PROGRAM stopping_mode
VAR
	ed_routine_stopping_idle: BOOL;
	stack_power_enabled: BOOL;
	RECTIFIER_OUTPUT_OFF: BOOL;// ADD LOGIC FOR MONITORING RECTIFIER OUTPUT - USE CT? VERIFY PS DOES NOT MOVE CURRENT WHEN POWERED OFF
	u_3112_b_stop_request: BOOL;
	u_3212_b_stop_request: BOOL;
	u_3312_b_stop_request: BOOL;
	u_3405_b_stop_request: BOOL;
	u_3160_b_stop_request: BOOL
;
	u_3260_b_stop_request: BOOL;
	u_3360_b_stop_request: BOOL;
	u_3370_b_stop_request: BOOL;
	u_3112_b_run_feedback: BOOL;
	u_3212_b_run_feedback: BOOL;
	u_3312_b_run_feedback: BOOL;
	u_3405_b_run_feedback: BOOL;
	u_3160_b_run_feedback: BOOL;
	u_3260_b_run_feedback: BOOL;
	u_3360_b_run_feedback: BOOL;
	u_3370_b_run_feedback: BOOL;
	
	nv_3110_b_stop_request:BOOL;
	av_3248_b_stop_request: BOOL;
	av_3148_b_stop_request: BOOL;
	nv_3335_b_stop_request: BOOL;
	nv_3235_b_stop_request: BOOL;
	nv_3135_b_stop_request: BOOL;
	nv_3310_b_stop_request: BOOL;
	nv_3210_b_stop_request: BOOL;
	ed_routine_stop_mode: BOOL;
	redox_doser_stop_request: BOOL;
	nv_3335_b_position_request: INT;
	av_3148_b_position_request: INT;
	av_3248_b_position_request: INT;
	ed_pumps_stopped: BOOL;

	nv_3335_b_position_feedback: INT;
	nv_3335_b_recycle_position: BOOL;
	av_3148_b_position_feedback: INT;
	av_3148_b_recycle_position: BOOL;
	av_3248_b_recycle_position: BOOL;
	ed_valves_stopped: BOOL;
	ed_stopped: BOOL;
	av_3348_b_position_request: INT;
	nv_3372_b_stop_request: BOOL;
	av_3348_b_position_feedback: INT;
	av_3348_b_recycle_position: BOOL;
	nv_3335_b_closed_feedback: BOOL;
	nv_3372_b_closed_feedback: BOOL;
	nv_3162_b_stop_request: BOOL;
	ed_critical_stop: BOOL;
	tmr_stop_pump_delay: TON;
	tmr_stop_pump_delay_pt: TIME := T#10S;
	tmr_stop_pump_delay_et: TIME;
	test_ramp: ramp;
	eng_test: BOOL;
	test_ramp_start_val: REAL;
	test_ramp_end_val: REAL;
	test_ramp_duration: INT;
END_VAR
VAR // added by the converter: edge detectors and wires of the graphical bodies
    _w1, _w2, _w3 : BOOL;
END_VAR

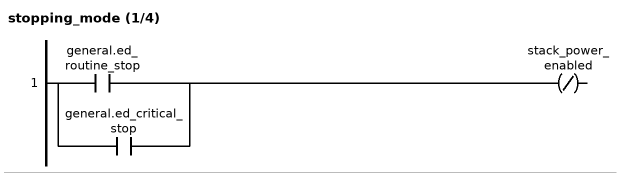
// NETWORK 1
stack_power_enabled := NOT (general.ed_routine_stop OR general.ed_critical_stop);

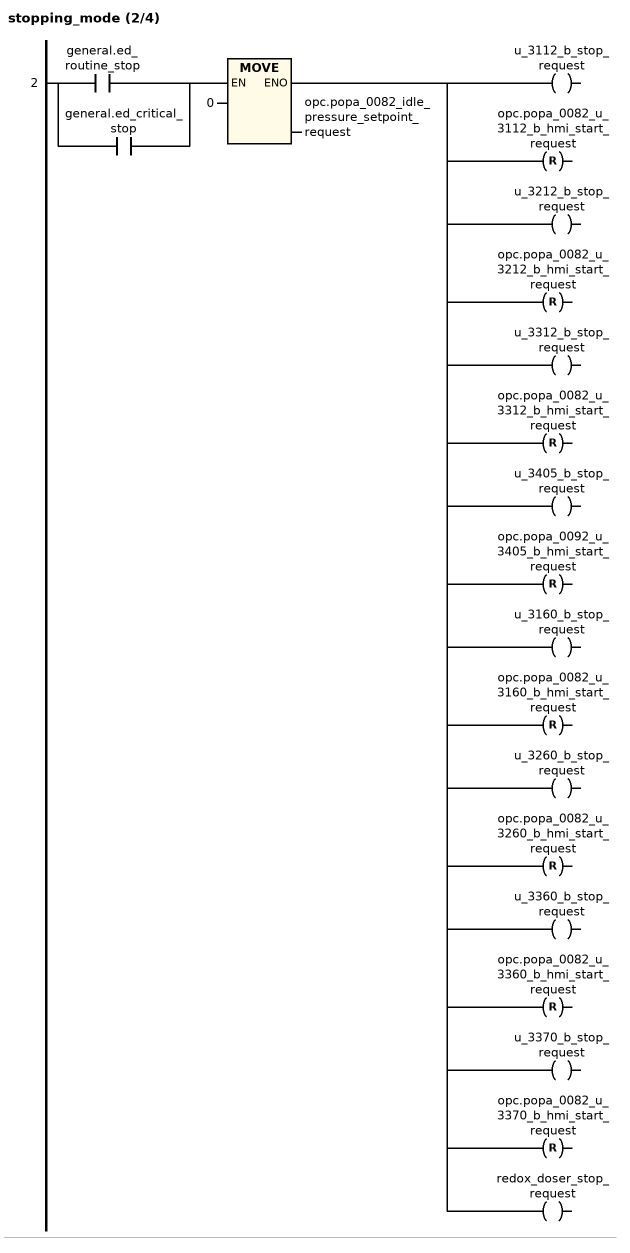
// NETWORK 2
_w1 := general.ed_routine_stop OR general.ed_critical_stop;
IF _w1 THEN opc.popa_0082_idle_pressure_setpoint_request := 0; END_IF
u_3112_b_stop_request := _w1;
opc.popa_0082_u_3112_b_hmi_start_request R= _w1;
u_3212_b_stop_request := _w1;
opc.popa_0082_u_3212_b_hmi_start_request R= _w1;
u_3312_b_stop_request := _w1;
opc.popa_0082_u_3312_b_hmi_start_request R= _w1;
u_3405_b_stop_request := _w1;
opc.popa_0092_u_3405_b_hmi_start_request R= _w1;
u_3160_b_stop_request := _w1;
opc.popa_0082_u_3160_b_hmi_start_request R= _w1;
u_3260_b_stop_request := _w1;
opc.popa_0082_u_3260_b_hmi_start_request R= _w1;
u_3360_b_stop_request := _w1;
opc.popa_0082_u_3360_b_hmi_start_request R= _w1;
u_3370_b_stop_request := _w1;
opc.popa_0082_u_3370_b_hmi_start_request R= _w1;
redox_doser_stop_request := _w1;

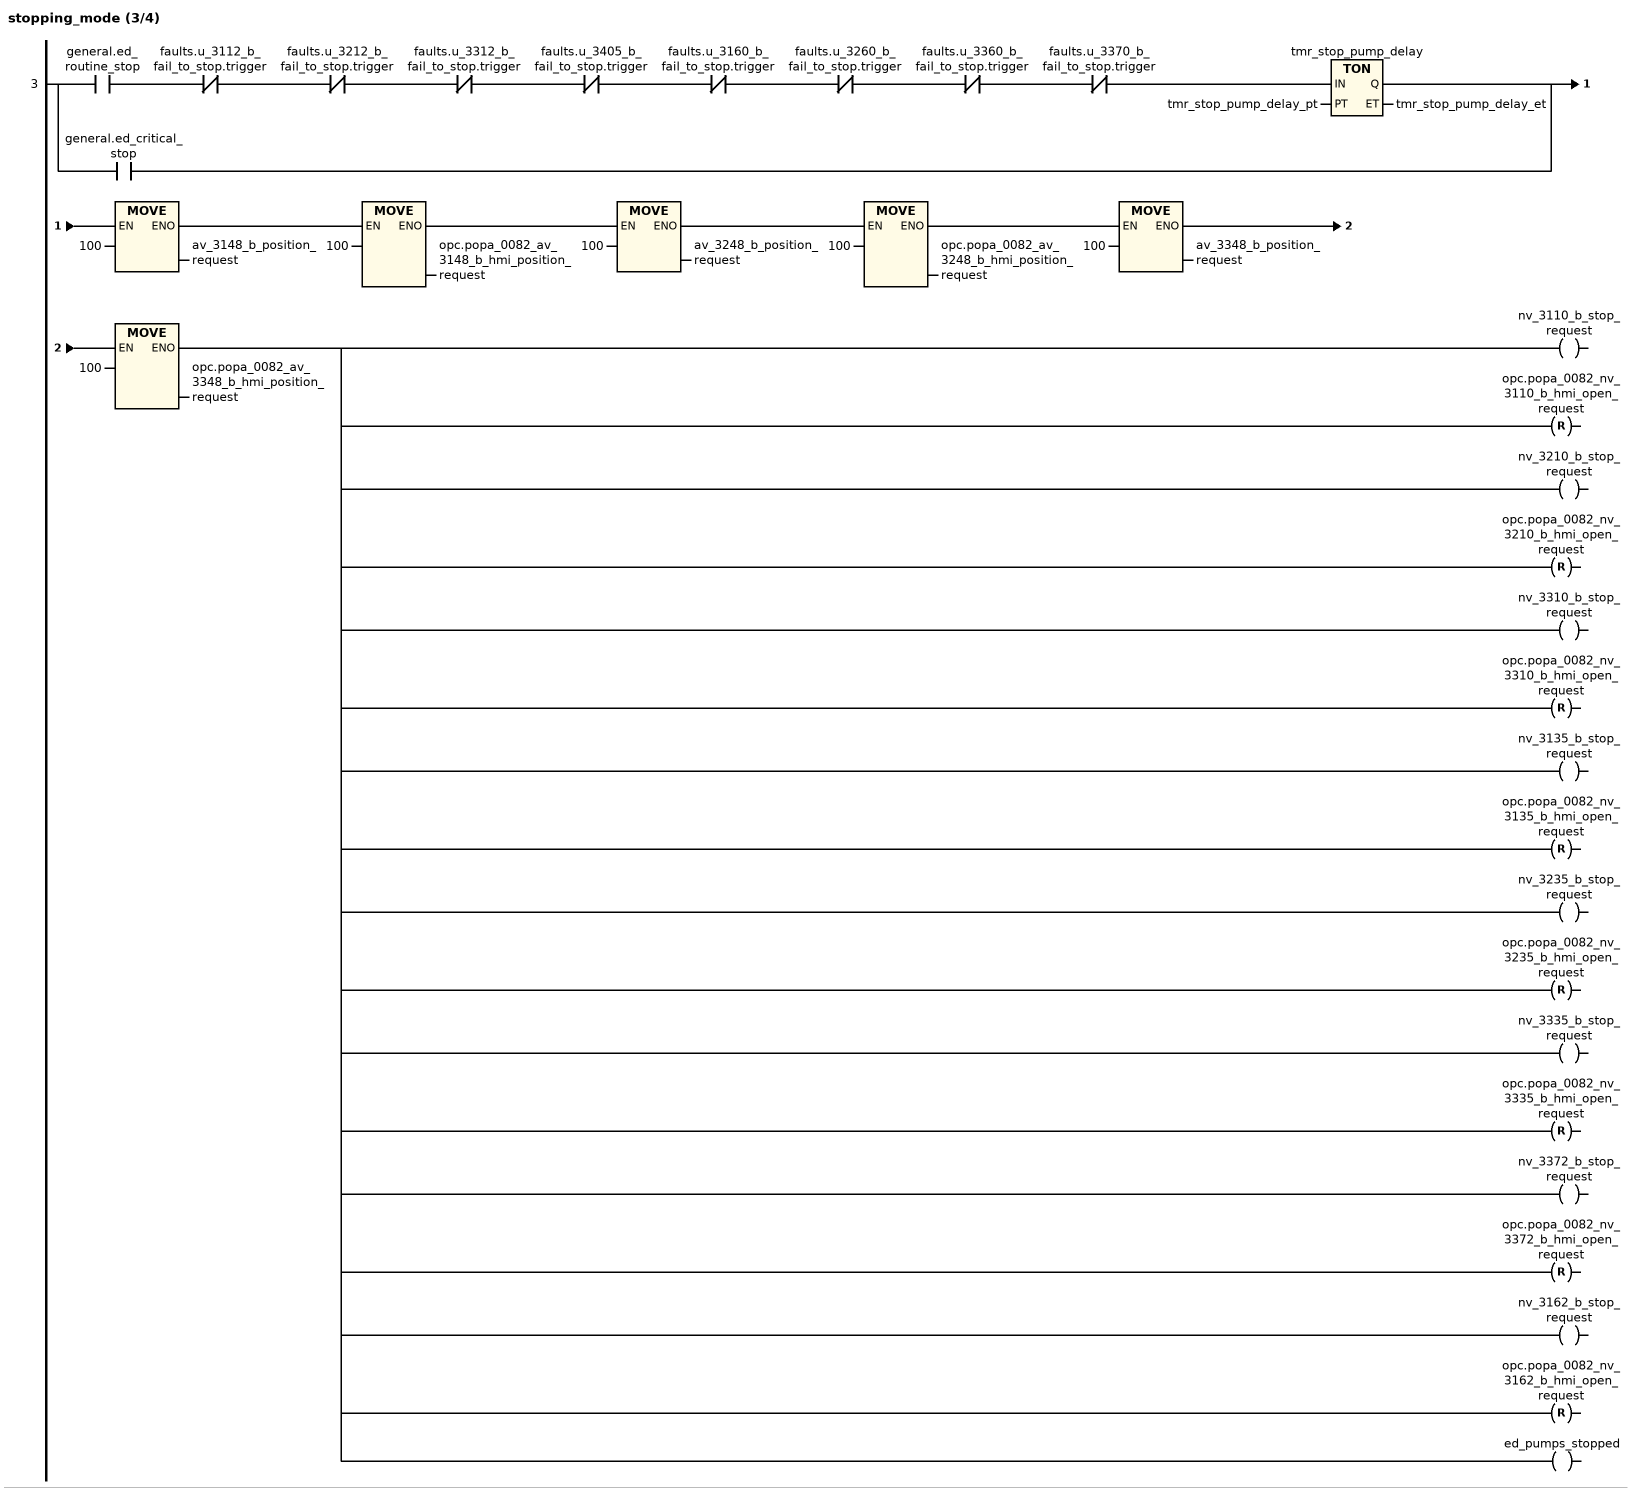
// NETWORK 3
tmr_stop_pump_delay(
    IN := general.ed_routine_stop AND NOT faults.u_3112_b_fail_to_stop.trigger AND NOT faults.u_3212_b_fail_to_stop.trigger AND NOT faults.u_3312_b_fail_to_stop.trigger AND NOT faults.u_3405_b_fail_to_stop.trigger AND NOT faults.u_3160_b_fail_to_stop.trigger AND NOT faults.u_3260_b_fail_to_stop.trigger AND NOT faults.u_3360_b_fail_to_stop.trigger AND NOT faults.u_3370_b_fail_to_stop.trigger,
    PT := tmr_stop_pump_delay_pt,
    ET => tmr_stop_pump_delay_et); // TON
_w2 := tmr_stop_pump_delay.Q OR general.ed_critical_stop;
IF _w2 THEN av_3148_b_position_request := 100; END_IF
IF _w2 THEN opc.popa_0082_av_3148_b_hmi_position_request := 100; END_IF
IF _w2 THEN av_3248_b_position_request := 100; END_IF
IF _w2 THEN opc.popa_0082_av_3248_b_hmi_position_request := 100; END_IF
IF _w2 THEN av_3348_b_position_request := 100; END_IF
IF _w2 THEN opc.popa_0082_av_3348_b_hmi_position_request := 100; END_IF
nv_3110_b_stop_request := _w2;
opc.popa_0082_nv_3110_b_hmi_open_request R= _w2;
nv_3210_b_stop_request := _w2;
opc.popa_0082_nv_3210_b_hmi_open_request R= _w2;
nv_3310_b_stop_request := _w2;
opc.popa_0082_nv_3310_b_hmi_open_request R= _w2;
nv_3135_b_stop_request := _w2;
opc.popa_0082_nv_3135_b_hmi_open_request R= _w2;
nv_3235_b_stop_request := _w2;
opc.popa_0082_nv_3235_b_hmi_open_request R= _w2;
nv_3335_b_stop_request := _w2;
opc.popa_0082_nv_3335_b_hmi_open_request R= _w2;
nv_3372_b_stop_request := _w2;
opc.popa_0082_nv_3372_b_hmi_open_request R= _w2;
nv_3162_b_stop_request := _w2;
opc.popa_0082_nv_3162_b_hmi_open_request R= _w2;
ed_pumps_stopped := _w2;

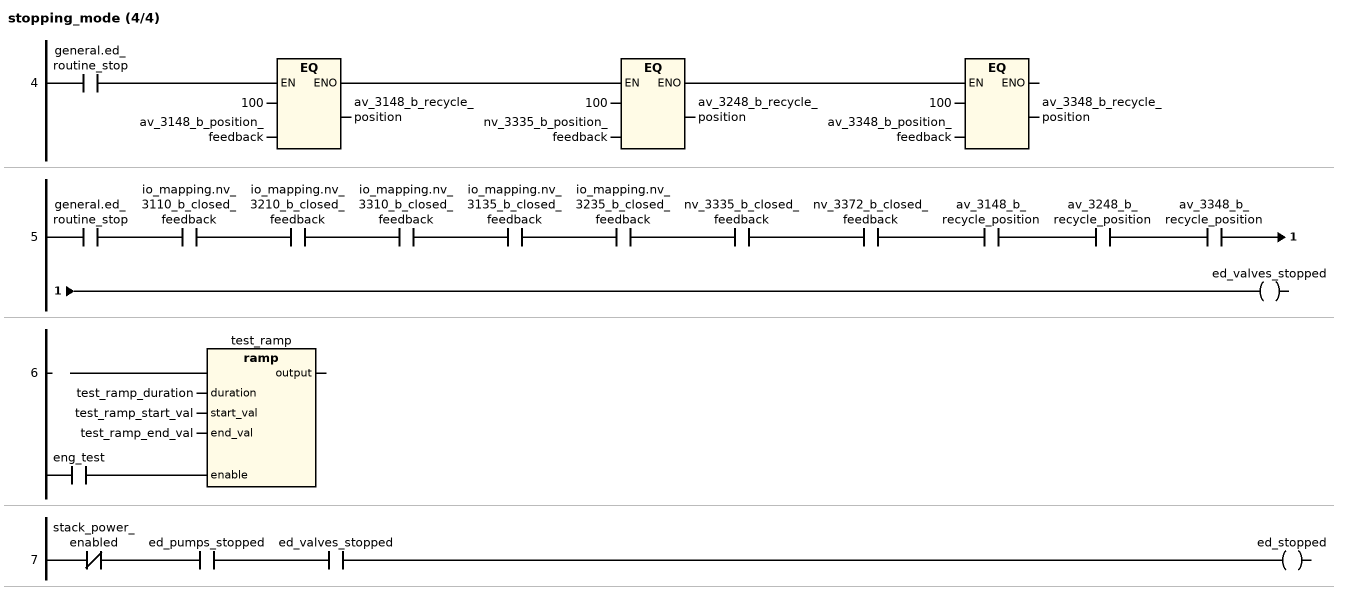
// NETWORK 4
_w3 := general.ed_routine_stop;
IF _w3 THEN av_3148_b_recycle_position := 100 = av_3148_b_position_feedback; END_IF
IF _w3 THEN av_3248_b_recycle_position := 100 = nv_3335_b_position_feedback; END_IF
IF _w3 THEN av_3348_b_recycle_position := 100 = av_3348_b_position_feedback; END_IF

// NETWORK 5
ed_valves_stopped := general.ed_routine_stop AND io_mapping.nv_3110_b_closed_feedback AND io_mapping.nv_3210_b_closed_feedback AND io_mapping.nv_3310_b_closed_feedback AND io_mapping.nv_3135_b_closed_feedback AND io_mapping.nv_3235_b_closed_feedback AND nv_3335_b_closed_feedback AND nv_3372_b_closed_feedback AND av_3148_b_recycle_position AND av_3248_b_recycle_position AND av_3348_b_recycle_position;

// NETWORK 6
test_ramp(
    duration := test_ramp_duration,
    start_val := test_ramp_start_val,
    end_val := test_ramp_end_val,
    enable := eng_test); // ramp

// NETWORK 7
ed_stopped := NOT stack_power_enabled AND ed_pumps_stopped AND ed_valves_stopped;

END_PROGRAM

(* stored: Version 1.1.0.1, ProductVersion 3.1.4024.15
   POU stopping_mode: Id {65ab387d-14b6-4597-8712-6f6f31d5a03f}, SpecialFunc None *)
